INTERFACE IPathQuery2

METHOD ToPosition : IPathQuery3
VAR_INPUT
  pos : LREAL;
END_VAR
END_METHOD

END_INTERFACE

(* stored: Version 1.1.0.1
   Itf IPathQuery2: Id {1d217fda-98d1-4876-be1b-73014b019343}
   Method ToPosition: Id {3b023a69-9ad7-4bd7-a98f-3e1429237ba0} *)
